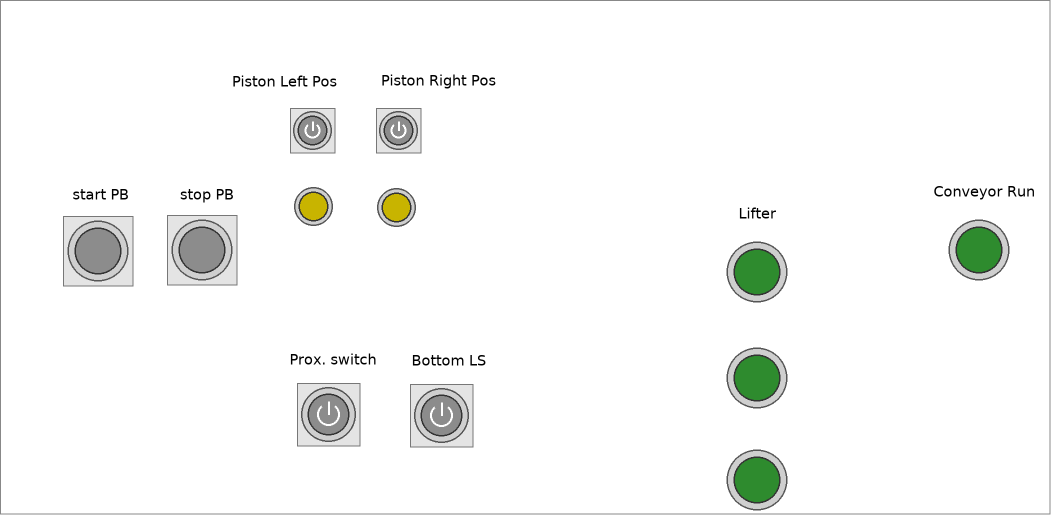
VISUALIZATION Visualization  // 1051x515
    PushSwitch (63,216 70x70), variable: MAIN.StartPB, behaviour: TAP, style: Switch-PushSwitch-Gray
    PushSwitch (167,215 70x70), variable: MAIN.StopPB, behaviour: TAP, style: Switch-PushSwitch-Gray
    PowerSwitch (297,381 63x67), variable: MAIN.ProxSwitch, behaviour: TOGGLE, style: Switch-PowerSwitch-Gray
    Lamp1 (944,215 70x70), variable: MAIN.ConveyorRun, style: Lamp-Lamp1-Green
    Lamp1 (722,237 70x70), variable: MAIN.LifterUp, style: Lamp-Lamp1-Green
    Lamp1 (722,343 70x70), variable: MAIN.LifterStop, style: Lamp-Lamp1-Green
    Label (50,174 102x41), "start PB"
    Label (156,174 102x41), "stop PB"
    Label (282,339 102x41), "Prox. switch"
    PowerSwitch (410,382 63x67), variable: MAIN.BottomLimitSwitch, behaviour: TOGGLE, style: Switch-PowerSwitch-Gray
    Label (398,340 102x41), "Bottom LS"
    PowerSwitch (290,103 45x55), variable: MAIN.PistonLeftPos, behaviour: TOGGLE, style: Switch-PowerSwitch-Gray
    PowerSwitch (376,103 45x55), variable: MAIN.PistonRightPos, behaviour: TOGGLE, style: Switch-PowerSwitch-Gray
    Label (222,61 125x41), "Piston Left Pos"
    Label (372,60 133x41), "Piston Right Pos"
    Label (918,171 133x41), "Conveyor Run"
    Lamp1 (722,445 70x70), variable: MAIN.LifterDown, style: Lamp-Lamp1-Green
    Label (691,193 133x41), "Lifter"
    Lamp1 (374,181 45x53), variable: MAIN.PistonMoveRight, style: Lamp-Lamp1-Yellow
    Lamp1 (291,180 45x53), variable: MAIN.PistonMoveLeft, style: Lamp-Lamp1-Yellow
END_VISUALIZATION

(* stored: Version 1.1.0.1, ProductVersion 3.1.4024.15
   Visu Visualization: Id {801d73d2-44be-4358-976c-36dc61e9cf90} *)
